// TIA Portal V16 export
// export: Created 2021-02-19T12:03:04.2794672Z, ExportSetting WithDefaults, DisplayName Totally Integrated Automation Portal, DisplayVersion V16 Update 3, DisplayName TIA Portal Version Control Interface, DisplayVersion V16 Update 2, DisplayName TIA Portal Openness, DisplayVersion V16 Update 3, DisplayName STEP 7 Professional, DisplayVersion V16 Update 3, DisplayName STEP 7 Safety, DisplayVersion V16, DisplayName WinCC Professional, DisplayVersion V16 Update 3
VAR_GLOBAL   // PLC tag table "PAL_TestFC18151"
   EventTrigger AT %M20.0 : Bool;
END_VAR
